(* IEC 61131-3 sources: ICSQuartz/benchmarks/oscat_basic_real_to_strf/src, 1 file *)

(* ---- program.st ---- *)
PROGRAM PLC_PRG
VAR_INPUT
    in_IN: REAL;
    in_N: INT;
    in_D: STRING;
END_VAR

REAL_TO_STRF(in_IN, in_N, in_D);

END_PROGRAM
